TYPE ST_PMLSubUnitInfo :
STRUCT
    bActive  : BOOL;
    eState   : E_PackMLState;
END_STRUCT
END_TYPE

(* stored: Version 1.1.0.1
   DUT ST_PMLSubUnitInfo: Id {1482e3c0-0723-4cff-92f7-18c9bee98f71} *)
